SYSTEM LandingGear
  (* Version 1.0, 2021-12-09, Fan *)
  APPLICATION LandingGearApp
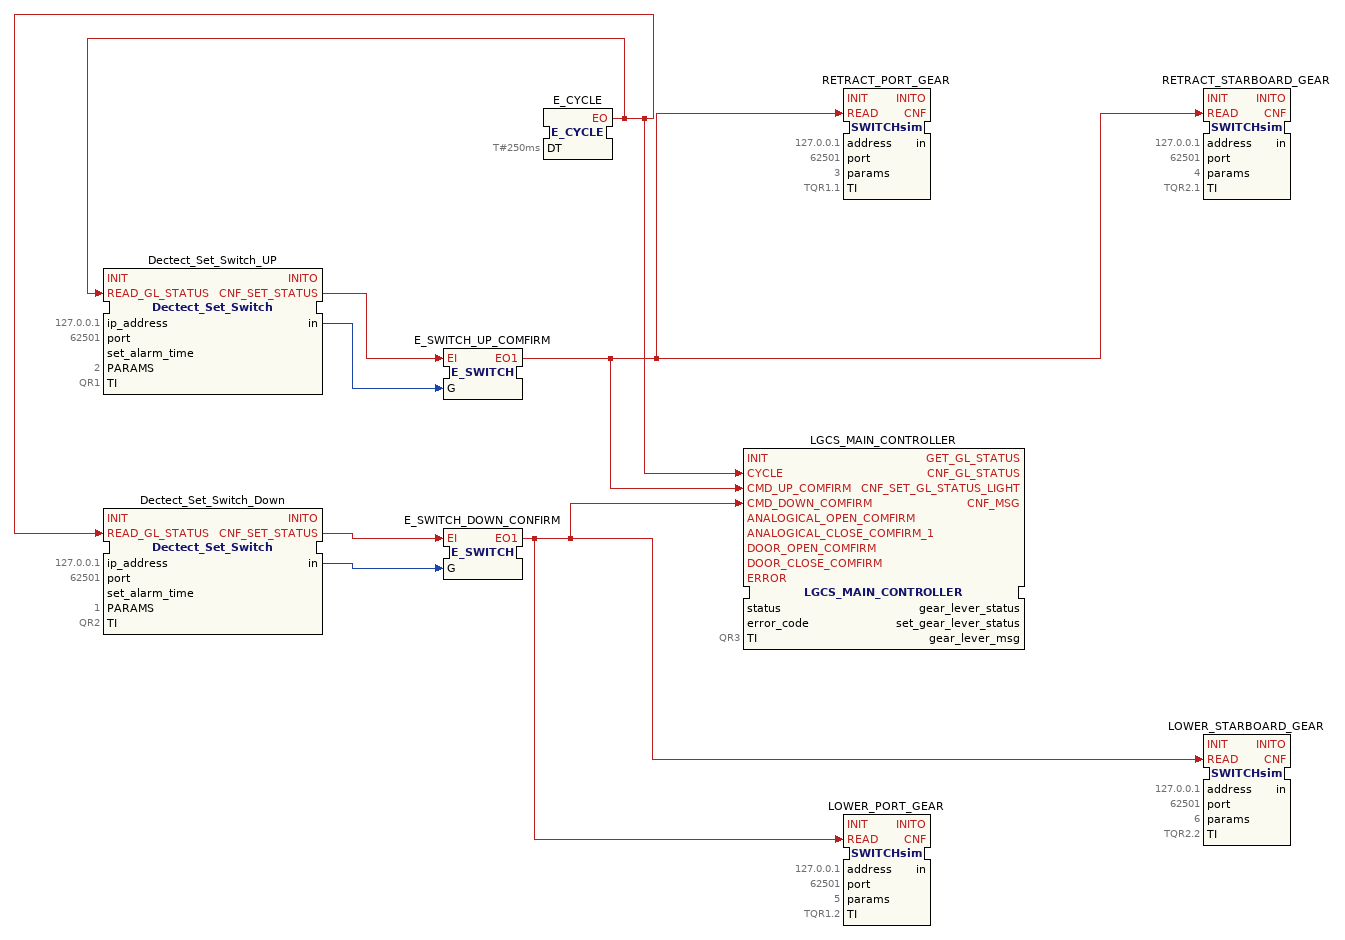
    FBS
      E_CYCLE : E_CYCLE(DT := T#250ms);
      Dectect_Set_Switch_UP : Dectect_Set_Switch(ip_address := 127.0.0.1, port := 62501, PARAMS := 2, TI := QR1);
      Dectect_Set_Switch_Down : Dectect_Set_Switch(ip_address := 127.0.0.1, port := 62501, PARAMS := 1, TI := QR2);
      E_SWITCH_UP_COMFIRM : E_SWITCH;
      E_SWITCH_DOWN_CONFIRM : E_SWITCH;
      LGCS_MAIN_CONTROLLER : LGCS_MAIN_CONTROLLER(TI := QR3);
      LOWER_PORT_GEAR : SWITCHsim(address := 127.0.0.1, port := 62501, params := 5, TI := TQR1.2);
      LOWER_STARBOARD_GEAR : SWITCHsim(address := 127.0.0.1, port := 62501, params := 6, TI := TQR2.2);
      RETRACT_PORT_GEAR : SWITCHsim(address := 127.0.0.1, port := 62501, params := 3, TI := TQR1.1);
      RETRACT_STARBOARD_GEAR : SWITCHsim(address := 127.0.0.1, port := 62501, params := 4, TI := TQR2.1);
    END_FBS
    EVENT_CONNECTIONS
      E_CYCLE.EO TO Dectect_Set_Switch_UP.READ_GL_STATUS;
      E_CYCLE.EO TO Dectect_Set_Switch_Down.READ_GL_STATUS;
      Dectect_Set_Switch_UP.CNF_SET_STATUS TO E_SWITCH_UP_COMFIRM.EI;
      E_CYCLE.EO TO LGCS_MAIN_CONTROLLER.CYCLE;
      E_SWITCH_UP_COMFIRM.EO1 TO LGCS_MAIN_CONTROLLER.CMD_UP_COMFIRM;
      E_SWITCH_DOWN_CONFIRM.EO1 TO LGCS_MAIN_CONTROLLER.CMD_DOWN_COMFIRM;
      Dectect_Set_Switch_Down.CNF_SET_STATUS TO E_SWITCH_DOWN_CONFIRM.EI;
      E_SWITCH_DOWN_CONFIRM.EO1 TO LOWER_PORT_GEAR.READ;
      E_SWITCH_DOWN_CONFIRM.EO1 TO LOWER_STARBOARD_GEAR.READ;
      E_SWITCH_UP_COMFIRM.EO1 TO RETRACT_PORT_GEAR.READ;
      E_SWITCH_UP_COMFIRM.EO1 TO RETRACT_STARBOARD_GEAR.READ;
    END_CONNECTIONS
    DATA_CONNECTIONS
      Dectect_Set_Switch_UP.in TO E_SWITCH_UP_COMFIRM.G;
      Dectect_Set_Switch_Down.in TO E_SWITCH_DOWN_CONFIRM.G;
    END_CONNECTIONS
  END_APPLICATION
  DEVICE FORTE_PC : FORTE_PC(MGR_ID := "localhost:61499")
    {SET_ATTRIBUTE(Profile, HOLOBLOC)} (* device profile *)
    RESOURCE EMB_RES : EMB_RES
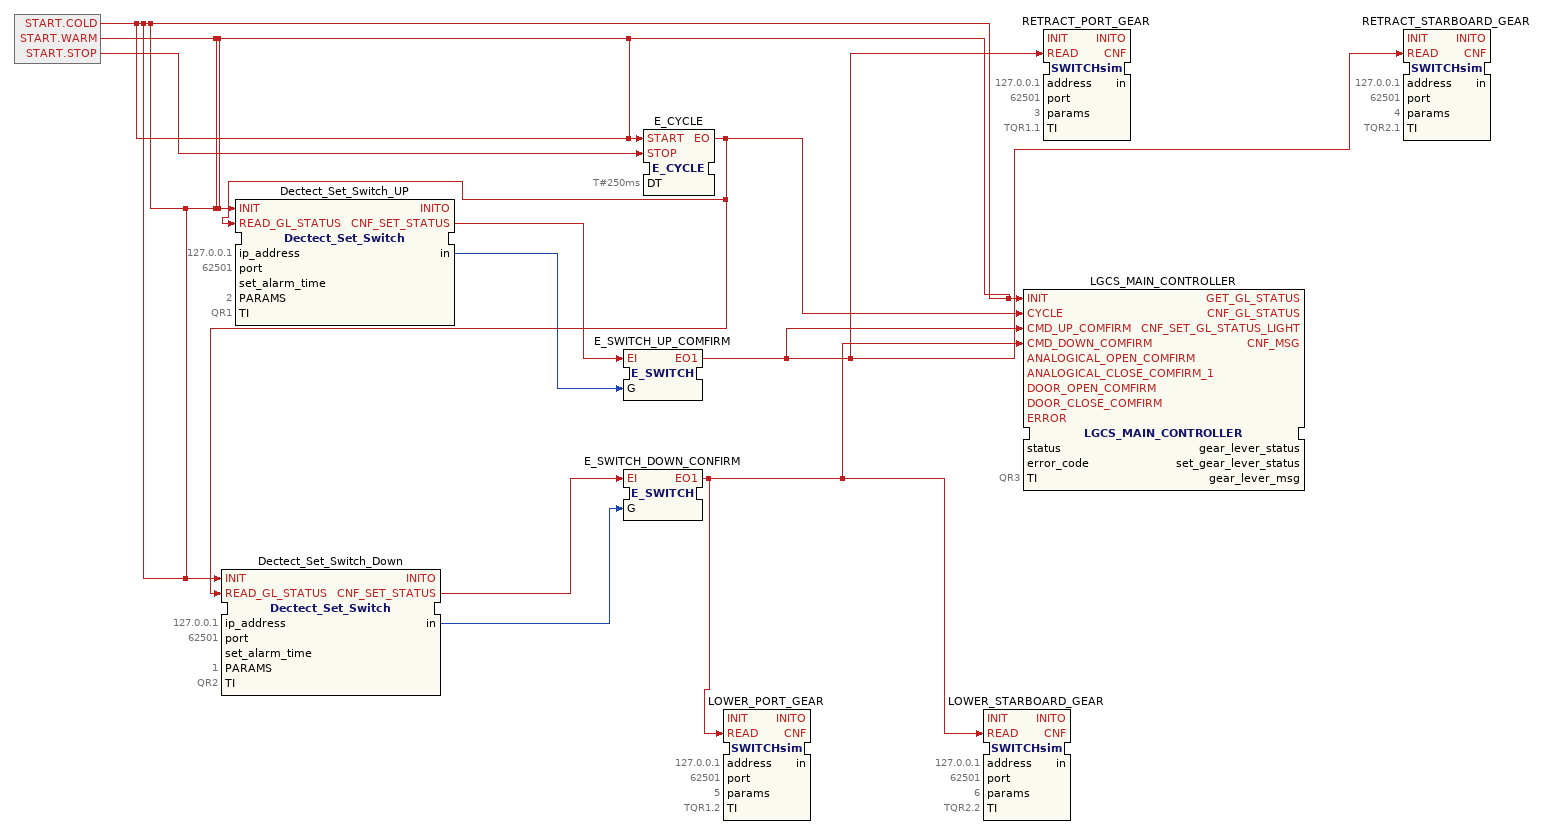
      FBS
        Dectect_Set_Switch_UP : Dectect_Set_Switch(ip_address := 127.0.0.1, port := 62501, PARAMS := 2, TI := QR1);
        Dectect_Set_Switch_Down : Dectect_Set_Switch(ip_address := 127.0.0.1, port := 62501, PARAMS := 1, TI := QR2);
        E_CYCLE : E_CYCLE(DT := T#250ms);
        E_SWITCH_UP_COMFIRM : E_SWITCH;
        E_SWITCH_DOWN_CONFIRM : E_SWITCH;
        LGCS_MAIN_CONTROLLER : LGCS_MAIN_CONTROLLER(TI := QR3);
        LOWER_PORT_GEAR : SWITCHsim(address := 127.0.0.1, port := 62501, params := 5, TI := TQR1.2);
        LOWER_STARBOARD_GEAR : SWITCHsim(address := 127.0.0.1, port := 62501, params := 6, TI := TQR2.2);
        RETRACT_PORT_GEAR : SWITCHsim(address := 127.0.0.1, port := 62501, params := 3, TI := TQR1.1);
        RETRACT_STARBOARD_GEAR : SWITCHsim(address := 127.0.0.1, port := 62501, params := 4, TI := TQR2.1);
      END_FBS
      EVENT_CONNECTIONS
        E_CYCLE.EO TO Dectect_Set_Switch_UP.READ_GL_STATUS;
        E_CYCLE.EO TO Dectect_Set_Switch_Down.READ_GL_STATUS;
        Dectect_Set_Switch_UP.CNF_SET_STATUS TO E_SWITCH_UP_COMFIRM.EI;
        START.COLD TO E_CYCLE.START;
        START.COLD TO Dectect_Set_Switch_Down.INIT;
        START.COLD TO Dectect_Set_Switch_UP.INIT;
        START.WARM TO Dectect_Set_Switch_UP.INIT;
        START.WARM TO Dectect_Set_Switch_Down.INIT;
        START.WARM TO E_CYCLE.START;
        START.STOP TO E_CYCLE.STOP;
        E_CYCLE.EO TO LGCS_MAIN_CONTROLLER.CYCLE;
        E_SWITCH_UP_COMFIRM.EO1 TO LGCS_MAIN_CONTROLLER.CMD_UP_COMFIRM;
        E_SWITCH_DOWN_CONFIRM.EO1 TO LGCS_MAIN_CONTROLLER.CMD_DOWN_COMFIRM;
        START.COLD TO LGCS_MAIN_CONTROLLER.INIT;
        START.WARM TO LGCS_MAIN_CONTROLLER.INIT;
        Dectect_Set_Switch_Down.CNF_SET_STATUS TO E_SWITCH_DOWN_CONFIRM.EI;
        E_SWITCH_DOWN_CONFIRM.EO1 TO LOWER_PORT_GEAR.READ;
        E_SWITCH_DOWN_CONFIRM.EO1 TO LOWER_STARBOARD_GEAR.READ;
        E_SWITCH_UP_COMFIRM.EO1 TO RETRACT_PORT_GEAR.READ;
        E_SWITCH_UP_COMFIRM.EO1 TO RETRACT_STARBOARD_GEAR.READ;
      END_CONNECTIONS
      DATA_CONNECTIONS
        Dectect_Set_Switch_UP.in TO E_SWITCH_UP_COMFIRM.G;
        Dectect_Set_Switch_Down.in TO E_SWITCH_DOWN_CONFIRM.G;
      END_CONNECTIONS
    END_RESOURCE
  END_DEVICE
  MAPPINGS
    LandingGearApp.Dectect_Set_Switch_UP ON FORTE_PC.EMB_RES.Dectect_Set_Switch_UP;
    LandingGearApp.Dectect_Set_Switch_Down ON FORTE_PC.EMB_RES.Dectect_Set_Switch_Down;
    LandingGearApp.E_CYCLE ON FORTE_PC.EMB_RES.E_CYCLE;
    LandingGearApp.E_SWITCH_UP_COMFIRM ON FORTE_PC.EMB_RES.E_SWITCH_UP_COMFIRM;
    LandingGearApp.E_SWITCH_DOWN_CONFIRM ON FORTE_PC.EMB_RES.E_SWITCH_DOWN_CONFIRM;
    LandingGearApp.LGCS_MAIN_CONTROLLER ON FORTE_PC.EMB_RES.LGCS_MAIN_CONTROLLER;
    LandingGearApp.LOWER_PORT_GEAR ON FORTE_PC.EMB_RES.LOWER_PORT_GEAR;
    LandingGearApp.LOWER_STARBOARD_GEAR ON FORTE_PC.EMB_RES.LOWER_STARBOARD_GEAR;
    LandingGearApp.RETRACT_PORT_GEAR ON FORTE_PC.EMB_RES.RETRACT_PORT_GEAR;
    LandingGearApp.RETRACT_STARBOARD_GEAR ON FORTE_PC.EMB_RES.RETRACT_STARBOARD_GEAR;
  END_MAPPINGS
  SEGMENTS
    Ethernet : Ethernet;
  END_SEGMENTS
  LINKS
    FORTE_PC => Ethernet;
  END_LINKS
END_SYSTEM
